PROGRAM CalibrationExperimentLoop
VAR
END_VAR

// Nothing
ADSLOGSTR(
	msgCtrlMask := ADSLOG_MSGTYPE_HINT, 
	msgFmtStr := 'Test message. Device is in calibration', 
	strArg := ''
);

END_PROGRAM

(* stored: Version 1.1.0.1, ProductVersion 3.1.4024.12
   POU CalibrationExperimentLoop: Id {e275cd2c-3601-4000-b109-c3a2be9dc278}, SpecialFunc None *)
